// TIA Portal V19 export
VAR_GLOBAL   // PLC tag table "D21"
   D21_Lp_EntryReq_LB322 AT %Q250.5 : Bool;   // 262SH1
   D21_Lp_SafetyReset_LB322 AT %Q250.6 : Bool;   // 262SH2
   D21_Pb_EntryReq_LB322 AT %I251.1 : Bool;   // 262SH1
   D21_Pb_SafetyReset_LB322 AT %I251.2 : Bool;   // 262SH2
   D21_Ls_Os1 AT %I1300.2 : Bool;   // 250DI2 - 262A1
   D21_Ls_Os2 AT %I1300.6 : Bool;   // 250DI6 - 262A1
   D21_Cancello_Chiuso AT %I250.7 : Bool;   // 26201
   D21_Cancello_Bloccato AT %I251.0 : Bool;   // 26003
   D21_Comando_Elettroserratura AT %Q250.4 : Bool;   // 26202
END_VAR
